FUNCTION_BLOCK PUBLIC FNB_Currentlvl
VAR_INPUT
	currentlevel : ARRAY [0..10] OF BOOL;
END_VAR
VAR_OUTPUT
	level :  INT;
END_VAR
VAR
	i :  INT;
END_VAR

(*aktuális szint beállítása*)
FOR i := 0 TO 10 DO
	IF currentlevel[i] THEN
		level := i;
		EXIT;
	END_IF
END_FOR

END_FUNCTION_BLOCK

(* stored: Version 1.1.0.1, ProductVersion 3.1.4024.15
   POU FNB_Currentlvl: Id {e19d7812-789a-426a-9e4a-db012e01589e}, SpecialFunc None *)
